{attribute 'pack_mode' := '3'}
{attribute 'ads-client-datatype-attribute' := 'example-datatype-value-ääö'}
//Test comment äääöö 
TYPE ST_TestDataType :
STRUCT
	Member : ST_Struct;
END_STRUCT
END_TYPE

(* stored: Version 1.1.0.1, ProductVersion 3.1.4024.12
   DUT ST_TestDataType: Id {6e01cb8a-1f0e-4e02-9cad-7b8e83b5dded} *)
